{attribute 'qualified_only'}
VAR_GLOBAL
	Axis_X		: AXIS_REF;
	Axis_Y		: AXIS_REF;
	Axis_Z		: AXIS_REF;
END_VAR

(* stored: Version 1.1.0.1, ProductVersion 3.1.4024.10
   GVL AXIS_Declaration: Id {f25a219c-e7dc-41e6-bca1-ceb9cdd45b48} *)
